TYPE ST_CFG_SIS_MsgManager_6_1 :
(**************************************************************************************
 * 	Application		:	BoxControl Framework
 *	Revision		:	$Revision: 404529 $
 *	Revision date	:	$Date: 2018-04-23 08:21:38 +0200 (Mo., 23 Apr 2018) $
 *	Last changed by	:	$Author: b7bolm $
 *	URL				:	$URL: http://almscdc.swisslog.com/repo/SWPD/Development/BoxControlFramework/20_Release/trunk/01_Software/BCF/BCF/JumpStart/20_Product/10_App/11_Com/10_Lib/10_Conv/12_MFCS/11_SIS/01_DUTs/11_SIS_6_1/ST_CFG_SIS_MsgManager_6_1.TcDUT $
 *
 *	Purpose			:	Configuration SIS V6.0
 *
 * ------------------------------------------------------------------------------------
 *	Copyright Swisslog [IP AG], Switzerland. All rights reserved.
 * 
 * ------------------------------------------------------------------------------------
 *	
 * 	Revision History: 
 *
 * 	VERSION			DATE			INITIALS			DESCRIPTION
 *	0.1				01.01.2001		swl					Example
 *
 **************************************************************************************)
STRUCT
	MFCS_Channel			: E_MFCS_Channel; // MFCS channel
	BufferLevelWarning		: UDINT; // Buffer warning
	BufferLevelAlarm		: UDINT; // Buffer alarm
	BufferLevelHysterese    : UDINT := 10; // Buffer level hysterese
	BaseDriver				: ST_CFG_SIS_BaseDriver; // Config base drive
	MirrorChannel			: E_MFCS_Channel; // Mirror channel
	Telegrams				: ST_SendTelegrams_6_1; // Telegram config
END_STRUCT
END_TYPE

(* stored: Version 1.1.0.1, ProductVersion 3.1.4022.12
   DUT ST_CFG_SIS_MsgManager_6_1: Id {be64321e-09c1-4ab1-9343-033ad2396c1c} *)
